FUNCTION_BLOCK basicHorimetro2 (* Basic Function Block Type - Horimetro com carga inicial dos valores persistidos *)
  (* Standard: 61499-2 *)
  (* Version 1.0.0, 11/05/2026, Hidryco, Hidryco, Corrige falha de restauracao apos reinicio do PLC. Expoe INIT_SEC/MIN/HOR para receber valores persistidos. *)
  PACKAGE Hidryco.HidrycoLib;
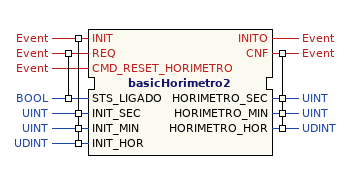
  EVENT_INPUT
    INIT WITH INIT_SEC, INIT_MIN, INIT_HOR; (* Inicializacao - carrega valores persistidos *)
    REQ WITH STS_LIGADO; (* Pulso de 1s para incrementar a contagem *)
    CMD_RESET_HORIMETRO; (* Zera o horimetro *)
  END_EVENT
  EVENT_OUTPUT
    INITO; (* Confirmacao de inicializacao *)
    CNF WITH HORIMETRO_SEC, HORIMETRO_MIN, HORIMETRO_HOR; (* Confirmacao de execucao *)
  END_EVENT
  VAR_INPUT
    STS_LIGADO : BOOL; (* 1 = equipamento em operacao (acumula tempo) *)
    INIT_SEC : UINT; (* Valor inicial de segundos (vindo do PERSISTENCE) *)
    INIT_MIN : UINT; (* Valor inicial de minutos (vindo do PERSISTENCE) *)
    INIT_HOR : UDINT; (* Valor inicial de horas (vindo do PERSISTENCE) *)
  END_VAR
  VAR_OUTPUT
    HORIMETRO_SEC : UINT; (* Segundos acumulados (0..59) *)
    HORIMETRO_MIN : UINT; (* Minutos acumulados (0..59) *)
    HORIMETRO_HOR : UDINT; (* Horas totais acumuladas *)
  END_VAR
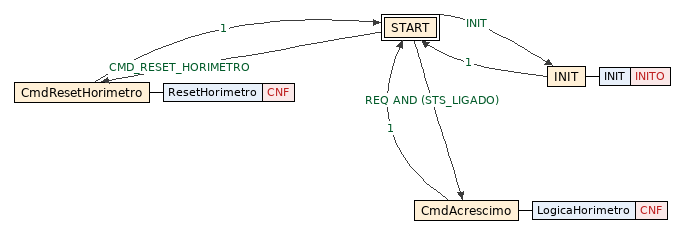
  EC_STATES
    START; (* Estado inicial *)
    INIT : INIT -> INITO; (* Inicializacao com valores persistidos *)
    CmdAcrescimo : LogicaHorimetro -> CNF; (* Incrementa contagem *)
    CmdResetHorimetro : ResetHorimetro -> CNF; (* Zera horimetro *)
  END_STATES
  EC_TRANSITIONS
    START TO INIT := INIT;
    INIT TO START := 1;
    START TO CmdAcrescimo := REQ AND (STS_LIGADO);
    CmdAcrescimo TO START := 1;
    START TO CmdResetHorimetro := CMD_RESET_HORIMETRO;
    CmdResetHorimetro TO START := 1;
  END_TRANSITIONS
  ALGORITHM INIT IN ST: (* Carrega valores persistidos apos boot/restart do PLC *)
// Restaura o estado do horimetro a partir dos valores lidos da persistencia.
// Sem isto, o horimetro reiniciaria do zero a cada reboot do PLC.
HORIMETRO_SEC := INIT_SEC;
HORIMETRO_MIN := INIT_MIN;
HORIMETRO_HOR := INIT_HOR;
  END_ALGORITHM
  ALGORITHM LogicaHorimetro IN ST: (* Incrementa segundos e propaga estouro para minutos e horas *)
// Incrementa 1 segundo a cada pulso REQ (esperado a 1 Hz) enquanto STS_LIGADO = TRUE
HORIMETRO_SEC := HORIMETRO_SEC + 1;

// Quando completa 60s, vira para o proximo minuto
IF (HORIMETRO_SEC >= 60) THEN
    HORIMETRO_MIN := HORIMETRO_MIN + 1;
    HORIMETRO_SEC := 0;
END_IF;

// Quando completa 60 min, vira para a proxima hora
IF (HORIMETRO_MIN >= 60) THEN
    HORIMETRO_HOR := HORIMETRO_HOR + 1;
    HORIMETRO_MIN := 0;
END_IF;
  END_ALGORITHM
  ALGORITHM ResetHorimetro IN ST: (* Zera todos os contadores *)
HORIMETRO_SEC := 0;
HORIMETRO_MIN := 0;
HORIMETRO_HOR := 0;
  END_ALGORITHM
END_FUNCTION_BLOCK
